PROGRAM Trend_sim
VAR
	//fbTrend		:FB_TrendLine;
	i : INT;
	iVal	:UDINT;
END_VAR

IF MAIN.bFirstCycle THEN
	FOR i := 1 TO 24 DO
		GV.aPoints[1,i].x := i;
		GV.aPoints[1,i].y := 1000;
		
		GV.aPoints[2,i].x := i;
		GV.aPoints[2,i].y := 50;
	END_FOR
END_IF

END_PROGRAM

(* stored: Version 1.1.0.1
   POU Trend_sim: Id {573151a2-82a4-46b0-93b4-82519825a2b1}, SpecialFunc None *)
